Fanuc KAREL source: kt00088.KL

-- PROVISIONAL review KL for V770-1; original PC SHA256 fe178912adb1b8b8c6e4141c2787d1f15a430688073278a401e47c71598641e7
-- Incomplete behavior may be omitted. Consult companion uncertainty JSON. Do not deploy.
PROGRAM KT00088
%NOLOCKGROUP
VAR
  OUT : REAL
-- UNRESOLVED_DECL Y1 type=002018
-- UNRESOLVED_DECL H2 type=002017
BEGIN
  -- UNRESOLVED_PC offsets 5-19; opcodes 2E,22,9D,33,B2
  -- UNRESOLVED_PC offsets 24-38; opcodes 2E,22,9D,33,B4
  -- UNRESOLVED_PC offsets 43-69; opcodes 22,9D,33,B1,22,9D,33,B3,54,64,23
  -- UNRESOLVED_PC offsets 74-78; opcodes 7F
END KT00088
